// Implicitly generated code : DO NOT EDIT
FUNCTION CheckRangeUnsigned : UDINT
VAR_INPUT
	value, lower, upper: UDINT;
END_VAR

{noflow}
IF (value < lower) THEN
	CheckRangeUnsigned := lower;
	F_Log(E_LogLevel.eFatal, 'Check UDINT range unsigned exception: {value} {lower} {upper}').WithLogger('CheckRangeUnsigned').WithAnyArg(value).WithAnyArg(lower).WithAnyArg(upper).CreateLog();
ELSIF(value > upper) THEN
	CheckRangeUnsigned := upper;
	F_Log(E_LogLevel.eFatal, 'Check UDINT range unsigned exception: {value} {lower} {upper}').WithLogger('CheckRangeUnsigned').WithAnyArg(value).WithAnyArg(lower).WithAnyArg(upper).CreateLog();
ELSE
	CheckRangeUnsigned := value;
END_IF
{flow}

END_FUNCTION

(* stored: Version 1.1.0.1, ProductVersion 3.1.4024.0
   POU CheckRangeUnsigned: Id {cded7342-7f00-4e95-a404-f3dedf2f50a8}, SpecialFunc CheckRangeUnsigned *)
